Fanuc KAREL source: kt00263.KL

-- PROVISIONAL review KL for V940-1; original PC SHA256 bde110919cbe1e484d64f9d8d52eade665a85db751ba479851a6bc5f9aedb6cf
-- Incomplete behavior may be omitted. Consult companion uncertainty JSON. Do not deploy.
PROGRAM KT00263
%NOLOCKGROUP
VAR
  R1 : REAL
  OUT : BOOLEAN
-- UNRESOLVED_DECL Y2 type=002018
BEGIN
  -- V9_ZERO_TABLE_METADATA_HINT layout=0001; no indexed target words; source/name/runtime held
  -- UNRESOLVED_PC offsets 5-16; opcodes 2E,23
  -- UNRESOLVED_PC offsets 21-35; opcodes 2E,22,9D,33,B2
  -- UNRESOLVED_PC offsets 40-63; opcodes 21,22,9D,33,B1,64,6D,23
  -- UNRESOLVED_PC offsets 68-72; opcodes 7F
END KT00263
